// TIA Portal V19 export
TYPE "LUC_typeInterlinkMode"
TITLE = LUC_typeInterlinkMode
// Link and unlink from parent module
// stored: Access Published
   STRUCT
      link : Bool;   // Command to link module to parent
      unlink : Bool;   // Command to unlink module from parent
      isLinked { ExternalWritable := 'False'} : Bool := true;   // Equipment module is linked to parent
   END_STRUCT;
END_TYPE
